// TIA Portal V17 export
// export: Created 2025-03-10T13:10:27.6830017Z, ExportSetting WithDefaults, DisplayName Totally Integrated Automation Portal, DisplayVersion V17 Update 8, DisplayName TIA Portal Openness, DisplayVersion V17 Update 8, DisplayName TIA Portal Version Control Interface, DisplayVersion V17, DisplayName SINAMICS Startdrive Advanced, DisplayVersion V17 SP2, DisplayName SINAMICS Startdrive G110M, G120, G120C, G120D, G120P, G115D, DisplayVersion V17 SP2, DisplayName SINAMICS Startdrive G130, G150, S120, S150, SINAMICS MV, S210, DisplayVersion V17 SP2, DisplayName STEP 7 Professional, DisplayVersion V17 Update 8, DisplayName SINUMERIK ONE STEP 7 Toolbox, DisplayVersion V17 Update 12, DisplayName SINUMERIK 840D sl STEP 7 Toolbox, DisplayVersion V17 Update 12, DisplayName STEP 7 Safety, DisplayVersion V17 Update 6, DisplayName WinCC Advanced, DisplayVersion V17 Update 8
FUNCTION "FC2106_SIGNAL_TOWER" : Void   // FC2106, LAD
{ S7_Optimized_Access := 'FALSE' }
AUTHOR : ETXETAR
VERSION : 1.0
// stored: AutoNumber false, IsIECCheckEnabled false, SetENOAutomatically false, UDAEnableTagReadback false
BEGIN

REGION Network 1: SIGNAL TOWER GREEN LIGHT OUTPUT / SIGNAL TOWER, GREEN LIGHT
   // GREEN LIGHT
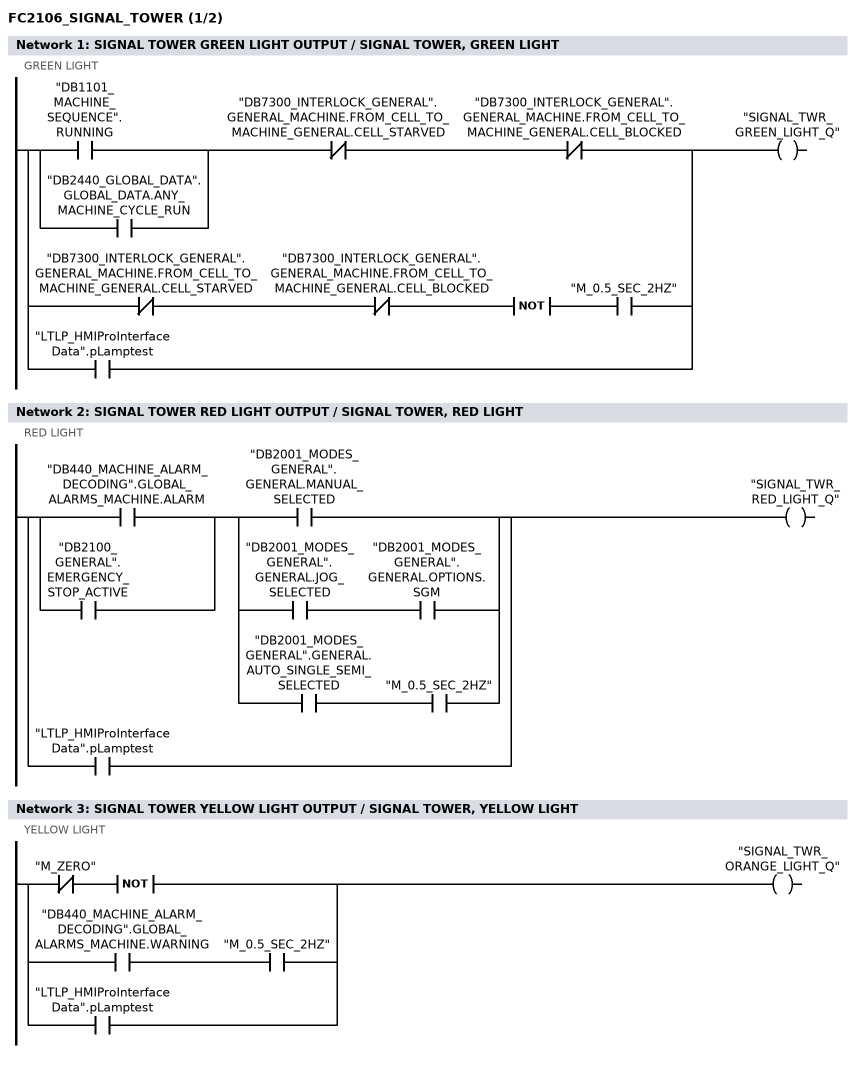
   RUNG wire#powerrail
      Contact( "DB1101_MACHINE_SEQUENCE".RUNNING )
      wire#w1
      I_Contact( "DB7300_INTERLOCK_GENERAL".GENERAL_MACHINE.FROM_CELL_TO_MACHINE_GENERAL.CELL_STARVED )
      I_Contact( "DB7300_INTERLOCK_GENERAL".GENERAL_MACHINE.FROM_CELL_TO_MACHINE_GENERAL.CELL_BLOCKED )
      wire#w2
      Coil( "SIGNAL_TWR_GREEN_LIGHT_Q" )
   END_RUNG
   RUNG wire#powerrail
      Contact( "DB2440_GLOBAL_DATA".GLOBAL_DATA.ANY_MACHINE_CYCLE_RUN )
   END_RUNG wire#w1
   RUNG wire#powerrail
      I_Contact( "DB7300_INTERLOCK_GENERAL".GENERAL_MACHINE.FROM_CELL_TO_MACHINE_GENERAL.CELL_STARVED )
      I_Contact( "DB7300_INTERLOCK_GENERAL".GENERAL_MACHINE.FROM_CELL_TO_MACHINE_GENERAL.CELL_BLOCKED )
      Not()
      Contact( "M_0.5_SEC_2HZ" )
   END_RUNG wire#w2
   RUNG wire#powerrail
      Contact( "LTLP_HMIProInterfaceData".pLamptest )
   END_RUNG wire#w2
   // the same network as SCL:
   "SIGNAL_TWR_GREEN_LIGHT_Q" := (("DB1101_MACHINE_SEQUENCE".RUNNING OR "DB2440_GLOBAL_DATA".GLOBAL_DATA.ANY_MACHINE_CYCLE_RUN) AND NOT "DB7300_INTERLOCK_GENERAL".GENERAL_MACHINE.FROM_CELL_TO_MACHINE_GENERAL.CELL_STARVED AND NOT "DB7300_INTERLOCK_GENERAL".GENERAL_MACHINE.FROM_CELL_TO_MACHINE_GENERAL.CELL_BLOCKED) OR (NOT (NOT "DB7300_INTERLOCK_GENERAL".GENERAL_MACHINE.FROM_CELL_TO_MACHINE_GENERAL.CELL_STARVED AND NOT "DB7300_INTERLOCK_GENERAL".GENERAL_MACHINE.FROM_CELL_TO_MACHINE_GENERAL.CELL_BLOCKED) AND "M_0.5_SEC_2HZ") OR "LTLP_HMIProInterfaceData".pLamptest;
END_REGION

REGION Network 2: SIGNAL TOWER RED LIGHT OUTPUT / SIGNAL TOWER, RED LIGHT
   // RED LIGHT
   RUNG wire#powerrail
      Contact( "DB440_MACHINE_ALARM_DECODING".GLOBAL_ALARMS_MACHINE.ALARM )
      wire#w1
      Contact( "DB2001_MODES_GENERAL".GENERAL.MANUAL_SELECTED )
      wire#w2
      Coil( "SIGNAL_TWR_RED_LIGHT_Q" )
   END_RUNG
   RUNG wire#powerrail
      Contact( "DB2100_GENERAL".EMERGENCY_STOP_ACTIVE )
   END_RUNG wire#w1
   RUNG wire#w1
      Contact( "DB2001_MODES_GENERAL".GENERAL.JOG_SELECTED )
      Contact( "DB2001_MODES_GENERAL".GENERAL.OPTIONS.SGM )
   END_RUNG wire#w2
   RUNG wire#w1
      Contact( "DB2001_MODES_GENERAL".GENERAL.AUTO_SINGLE_SEMI_SELECTED )
      Contact( "M_0.5_SEC_2HZ" )
   END_RUNG wire#w2
   RUNG wire#powerrail
      Contact( "LTLP_HMIProInterfaceData".pLamptest )
   END_RUNG wire#w2
   // the same network as SCL:
   "SIGNAL_TWR_RED_LIGHT_Q" := (("DB440_MACHINE_ALARM_DECODING".GLOBAL_ALARMS_MACHINE.ALARM OR "DB2100_GENERAL".EMERGENCY_STOP_ACTIVE) AND ("DB2001_MODES_GENERAL".GENERAL.MANUAL_SELECTED OR ("DB2001_MODES_GENERAL".GENERAL.JOG_SELECTED AND "DB2001_MODES_GENERAL".GENERAL.OPTIONS.SGM) OR ("DB2001_MODES_GENERAL".GENERAL.AUTO_SINGLE_SEMI_SELECTED AND "M_0.5_SEC_2HZ"))) OR "LTLP_HMIProInterfaceData".pLamptest;
END_REGION

REGION Network 3: SIGNAL TOWER YELLOW LIGHT OUTPUT / SIGNAL TOWER, YELLOW LIGHT
   // YELLOW LIGHT
   RUNG wire#powerrail
      I_Contact( "M_ZERO" )
      Not()
      wire#w1
      Coil( "SIGNAL_TWR_ORANGE_LIGHT_Q" )
   END_RUNG
   RUNG wire#powerrail
      Contact( "DB440_MACHINE_ALARM_DECODING".GLOBAL_ALARMS_MACHINE.WARNING )
      Contact( "M_0.5_SEC_2HZ" )
   END_RUNG wire#w1
   RUNG wire#powerrail
      Contact( "LTLP_HMIProInterfaceData".pLamptest )
   END_RUNG wire#w1
   // the same network as SCL:
   "SIGNAL_TWR_ORANGE_LIGHT_Q" := NOT (NOT "M_ZERO") OR ("DB440_MACHINE_ALARM_DECODING".GLOBAL_ALARMS_MACHINE.WARNING AND "M_0.5_SEC_2HZ") OR "LTLP_HMIProInterfaceData".pLamptest;
END_REGION

REGION Network 4: SIGNAL TOWER BLUE LIGHT OUTPUT / SIGNAL TOWER, BLUE LED
   // Blue Light
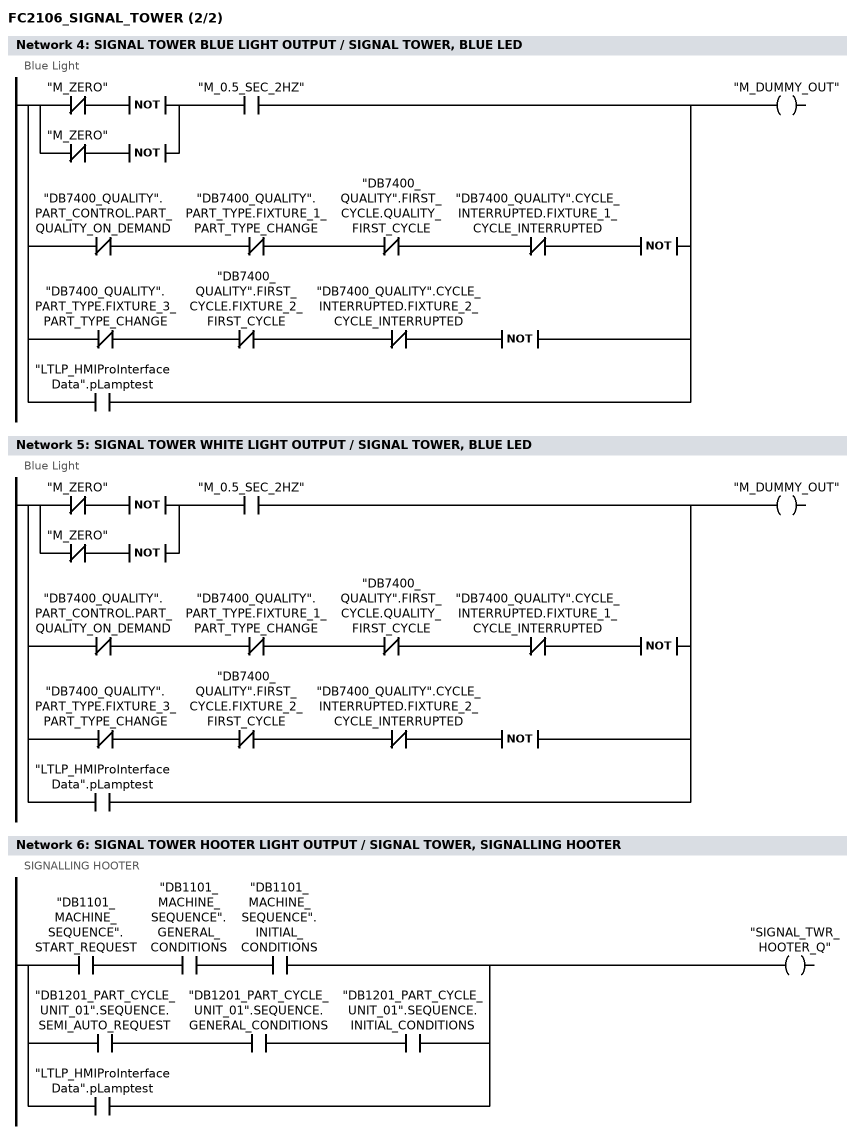
   RUNG wire#powerrail
      I_Contact( "M_ZERO" )
      Not()
      wire#w1
      Contact( "M_0.5_SEC_2HZ" )
      wire#w2
      Coil( "M_DUMMY_OUT" )
   END_RUNG
   RUNG wire#powerrail
      I_Contact( "M_ZERO" )
      Not()
   END_RUNG wire#w1
   RUNG wire#powerrail
      I_Contact( "DB7400_QUALITY".PART_CONTROL.PART_QUALITY_ON_DEMAND )
      I_Contact( "DB7400_QUALITY".PART_TYPE.FIXTURE_1_PART_TYPE_CHANGE )
      I_Contact( "DB7400_QUALITY".FIRST_CYCLE.QUALITY_FIRST_CYCLE )
      I_Contact( "DB7400_QUALITY".CYCLE_INTERRUPTED.FIXTURE_1_CYCLE_INTERRUPTED )
      Not()
   END_RUNG wire#w2
   RUNG wire#powerrail
      I_Contact( "DB7400_QUALITY".PART_TYPE.FIXTURE_3_PART_TYPE_CHANGE )
      I_Contact( "DB7400_QUALITY".FIRST_CYCLE.FIXTURE_2_FIRST_CYCLE )
      I_Contact( "DB7400_QUALITY".CYCLE_INTERRUPTED.FIXTURE_2_CYCLE_INTERRUPTED )
      Not()
   END_RUNG wire#w2
   RUNG wire#powerrail
      Contact( "LTLP_HMIProInterfaceData".pLamptest )
   END_RUNG wire#w2
   // the same network as SCL:
   "M_DUMMY_OUT" := ((NOT (NOT "M_ZERO") OR NOT (NOT "M_ZERO")) AND "M_0.5_SEC_2HZ") OR NOT (NOT "DB7400_QUALITY".PART_CONTROL.PART_QUALITY_ON_DEMAND AND NOT "DB7400_QUALITY".PART_TYPE.FIXTURE_1_PART_TYPE_CHANGE AND NOT "DB7400_QUALITY".FIRST_CYCLE.QUALITY_FIRST_CYCLE AND NOT "DB7400_QUALITY".CYCLE_INTERRUPTED.FIXTURE_1_CYCLE_INTERRUPTED) OR NOT (NOT "DB7400_QUALITY".PART_TYPE.FIXTURE_3_PART_TYPE_CHANGE AND NOT "DB7400_QUALITY".FIRST_CYCLE.FIXTURE_2_FIRST_CYCLE AND NOT "DB7400_QUALITY".CYCLE_INTERRUPTED.FIXTURE_2_CYCLE_INTERRUPTED) OR "LTLP_HMIProInterfaceData".pLamptest;
END_REGION

REGION Network 5: SIGNAL TOWER WHITE LIGHT OUTPUT / SIGNAL TOWER, BLUE LED
   // Blue Light
   RUNG wire#powerrail
      I_Contact( "M_ZERO" )
      Not()
      wire#w1
      Contact( "M_0.5_SEC_2HZ" )
      wire#w2
      Coil( "M_DUMMY_OUT" )
   END_RUNG
   RUNG wire#powerrail
      I_Contact( "M_ZERO" )
      Not()
   END_RUNG wire#w1
   RUNG wire#powerrail
      I_Contact( "DB7400_QUALITY".PART_CONTROL.PART_QUALITY_ON_DEMAND )
      I_Contact( "DB7400_QUALITY".PART_TYPE.FIXTURE_1_PART_TYPE_CHANGE )
      I_Contact( "DB7400_QUALITY".FIRST_CYCLE.QUALITY_FIRST_CYCLE )
      I_Contact( "DB7400_QUALITY".CYCLE_INTERRUPTED.FIXTURE_1_CYCLE_INTERRUPTED )
      Not()
   END_RUNG wire#w2
   RUNG wire#powerrail
      I_Contact( "DB7400_QUALITY".PART_TYPE.FIXTURE_3_PART_TYPE_CHANGE )
      I_Contact( "DB7400_QUALITY".FIRST_CYCLE.FIXTURE_2_FIRST_CYCLE )
      I_Contact( "DB7400_QUALITY".CYCLE_INTERRUPTED.FIXTURE_2_CYCLE_INTERRUPTED )
      Not()
   END_RUNG wire#w2
   RUNG wire#powerrail
      Contact( "LTLP_HMIProInterfaceData".pLamptest )
   END_RUNG wire#w2
   // the same network as SCL:
   "M_DUMMY_OUT" := ((NOT (NOT "M_ZERO") OR NOT (NOT "M_ZERO")) AND "M_0.5_SEC_2HZ") OR NOT (NOT "DB7400_QUALITY".PART_CONTROL.PART_QUALITY_ON_DEMAND AND NOT "DB7400_QUALITY".PART_TYPE.FIXTURE_1_PART_TYPE_CHANGE AND NOT "DB7400_QUALITY".FIRST_CYCLE.QUALITY_FIRST_CYCLE AND NOT "DB7400_QUALITY".CYCLE_INTERRUPTED.FIXTURE_1_CYCLE_INTERRUPTED) OR NOT (NOT "DB7400_QUALITY".PART_TYPE.FIXTURE_3_PART_TYPE_CHANGE AND NOT "DB7400_QUALITY".FIRST_CYCLE.FIXTURE_2_FIRST_CYCLE AND NOT "DB7400_QUALITY".CYCLE_INTERRUPTED.FIXTURE_2_CYCLE_INTERRUPTED) OR "LTLP_HMIProInterfaceData".pLamptest;
END_REGION

REGION Network 6: SIGNAL TOWER HOOTER LIGHT OUTPUT / SIGNAL TOWER, SIGNALLING HOOTER
   // SIGNALLING HOOTER
   RUNG wire#powerrail
      Contact( "DB1101_MACHINE_SEQUENCE".START_REQUEST )
      Contact( "DB1101_MACHINE_SEQUENCE".GENERAL_CONDITIONS )
      Contact( "DB1101_MACHINE_SEQUENCE".INITIAL_CONDITIONS )
      wire#w1
      Coil( "SIGNAL_TWR_HOOTER_Q" )
   END_RUNG
   RUNG wire#powerrail
      Contact( "DB1201_PART_CYCLE_UNIT_01".SEQUENCE.SEMI_AUTO_REQUEST )
      Contact( "DB1201_PART_CYCLE_UNIT_01".SEQUENCE.GENERAL_CONDITIONS )
      Contact( "DB1201_PART_CYCLE_UNIT_01".SEQUENCE.INITIAL_CONDITIONS )
   END_RUNG wire#w1
   RUNG wire#powerrail
      Contact( "LTLP_HMIProInterfaceData".pLamptest )
   END_RUNG wire#w1
   // the same network as SCL:
   "SIGNAL_TWR_HOOTER_Q" := ("DB1101_MACHINE_SEQUENCE".START_REQUEST AND "DB1101_MACHINE_SEQUENCE".GENERAL_CONDITIONS AND "DB1101_MACHINE_SEQUENCE".INITIAL_CONDITIONS) OR ("DB1201_PART_CYCLE_UNIT_01".SEQUENCE.SEMI_AUTO_REQUEST AND "DB1201_PART_CYCLE_UNIT_01".SEQUENCE.GENERAL_CONDITIONS AND "DB1201_PART_CYCLE_UNIT_01".SEQUENCE.INITIAL_CONDITIONS) OR "LTLP_HMIProInterfaceData".pLamptest;
END_REGION
END_FUNCTION
